(* IEC 61131-3 sources: TA/Tests/RetainTest/OLD/FBtest (part 4) *)

    ARRAY_LWORD_OUT_AUTO_2[0] := ARRAY_LWORD_OUT_AUTO_1[0];
    ARRAY_LWORD_OUT_AUTO_2[1] := ARRAY_LWORD_OUT_AUTO_1[1];
    ARRAY_LWORD_OUT_AUTO_2[2] := ARRAY_LWORD_OUT_AUTO_1[2];
    ARRAY_LWORD_OUT_AUTO_2[3] := ARRAY_LWORD_OUT_AUTO_1[3];
    ARRAY_LWORD_OUT_AUTO_2[4] := ARRAY_LWORD_OUT_AUTO_1[4];
    ARRAY_LWORD_OUT_AUTO_2[5] := ARRAY_LWORD_OUT_AUTO_1[5];
    ARRAY_LWORD_OUT_AUTO_2[6] := ARRAY_LWORD_OUT_AUTO_1[6];
    ARRAY_LWORD_OUT_AUTO_2[7] := ARRAY_LWORD_OUT_AUTO_1[7];
    ARRAY_LWORD_OUT_AUTO_2[8] := ARRAY_LWORD_OUT_AUTO_1[8];
    ARRAY_LWORD_OUT_AUTO_2[9] := ARRAY_LWORD_OUT_AUTO_1[9];

    ARRAY_REAL_OUT_AUTO_2[0] := ARRAY_REAL_OUT_AUTO_1[0];
    ARRAY_REAL_OUT_AUTO_2[1] := ARRAY_REAL_OUT_AUTO_1[1];
    ARRAY_REAL_OUT_AUTO_2[2] := ARRAY_REAL_OUT_AUTO_1[2];
    ARRAY_REAL_OUT_AUTO_2[3] := ARRAY_REAL_OUT_AUTO_1[3];
    ARRAY_REAL_OUT_AUTO_2[4] := ARRAY_REAL_OUT_AUTO_1[4];
    ARRAY_REAL_OUT_AUTO_2[5] := ARRAY_REAL_OUT_AUTO_1[5];
    ARRAY_REAL_OUT_AUTO_2[6] := ARRAY_REAL_OUT_AUTO_1[6];
    ARRAY_REAL_OUT_AUTO_2[7] := ARRAY_REAL_OUT_AUTO_1[7];
    ARRAY_REAL_OUT_AUTO_2[8] := ARRAY_REAL_OUT_AUTO_1[8];
    ARRAY_REAL_OUT_AUTO_2[9] := ARRAY_REAL_OUT_AUTO_1[9];

    ARRAY_SINT_OUT_AUTO_2[0] := ARRAY_SINT_OUT_AUTO_1[0];
    ARRAY_SINT_OUT_AUTO_2[1] := ARRAY_SINT_OUT_AUTO_1[1];
    ARRAY_SINT_OUT_AUTO_2[2] := ARRAY_SINT_OUT_AUTO_1[2];
    ARRAY_SINT_OUT_AUTO_2[3] := ARRAY_SINT_OUT_AUTO_1[3];
    ARRAY_SINT_OUT_AUTO_2[4] := ARRAY_SINT_OUT_AUTO_1[4];
    ARRAY_SINT_OUT_AUTO_2[5] := ARRAY_SINT_OUT_AUTO_1[5];
    ARRAY_SINT_OUT_AUTO_2[6] := ARRAY_SINT_OUT_AUTO_1[6];
    ARRAY_SINT_OUT_AUTO_2[7] := ARRAY_SINT_OUT_AUTO_1[7];
    ARRAY_SINT_OUT_AUTO_2[8] := ARRAY_SINT_OUT_AUTO_1[8];
    ARRAY_SINT_OUT_AUTO_2[9] := ARRAY_SINT_OUT_AUTO_1[9];

    ARRAY_STRING_OUT_AUTO_2[0] := ARRAY_STRING_OUT_AUTO_1[0];
    ARRAY_STRING_OUT_AUTO_2[1] := ARRAY_STRING_OUT_AUTO_1[1];
    ARRAY_STRING_OUT_AUTO_2[2] := ARRAY_STRING_OUT_AUTO_1[2];
    ARRAY_STRING_OUT_AUTO_2[3] := ARRAY_STRING_OUT_AUTO_1[3];
    ARRAY_STRING_OUT_AUTO_2[4] := ARRAY_STRING_OUT_AUTO_1[4];
    ARRAY_STRING_OUT_AUTO_2[5] := ARRAY_STRING_OUT_AUTO_1[5];
    ARRAY_STRING_OUT_AUTO_2[6] := ARRAY_STRING_OUT_AUTO_1[6];
    ARRAY_STRING_OUT_AUTO_2[7] := ARRAY_STRING_OUT_AUTO_1[7];
    ARRAY_STRING_OUT_AUTO_2[8] := ARRAY_STRING_OUT_AUTO_1[8];
    ARRAY_STRING_OUT_AUTO_2[9] := ARRAY_STRING_OUT_AUTO_1[9];

    ARRAY_TIME_OUT_AUTO_2[0] := ARRAY_TIME_OUT_AUTO_1[0];
    ARRAY_TIME_OUT_AUTO_2[1] := ARRAY_TIME_OUT_AUTO_1[1];
    ARRAY_TIME_OUT_AUTO_2[2] := ARRAY_TIME_OUT_AUTO_1[2];
    ARRAY_TIME_OUT_AUTO_2[3] := ARRAY_TIME_OUT_AUTO_1[3];
    ARRAY_TIME_OUT_AUTO_2[4] := ARRAY_TIME_OUT_AUTO_1[4];
    ARRAY_TIME_OUT_AUTO_2[5] := ARRAY_TIME_OUT_AUTO_1[5];
    ARRAY_TIME_OUT_AUTO_2[6] := ARRAY_TIME_OUT_AUTO_1[6];
    ARRAY_TIME_OUT_AUTO_2[7] := ARRAY_TIME_OUT_AUTO_1[7];
    ARRAY_TIME_OUT_AUTO_2[8] := ARRAY_TIME_OUT_AUTO_1[8];
    ARRAY_TIME_OUT_AUTO_2[9] := ARRAY_TIME_OUT_AUTO_1[9];

    ARRAY_UDINT_OUT_AUTO_2[0] := ARRAY_UDINT_OUT_AUTO_1[0];
    ARRAY_UDINT_OUT_AUTO_2[1] := ARRAY_UDINT_OUT_AUTO_1[1];
    ARRAY_UDINT_OUT_AUTO_2[2] := ARRAY_UDINT_OUT_AUTO_1[2];
    ARRAY_UDINT_OUT_AUTO_2[3] := ARRAY_UDINT_OUT_AUTO_1[3];
    ARRAY_UDINT_OUT_AUTO_2[4] := ARRAY_UDINT_OUT_AUTO_1[4];
    ARRAY_UDINT_OUT_AUTO_2[5] := ARRAY_UDINT_OUT_AUTO_1[5];
    ARRAY_UDINT_OUT_AUTO_2[6] := ARRAY_UDINT_OUT_AUTO_1[6];
    ARRAY_UDINT_OUT_AUTO_2[7] := ARRAY_UDINT_OUT_AUTO_1[7];
    ARRAY_UDINT_OUT_AUTO_2[8] := ARRAY_UDINT_OUT_AUTO_1[6];
    ARRAY_UDINT_OUT_AUTO_2[9] := ARRAY_UDINT_OUT_AUTO_1[7];

    ARRAY_UINT_OUT_AUTO_2[0] := ARRAY_UINT_OUT_AUTO_1[0];
    ARRAY_UINT_OUT_AUTO_2[1] := ARRAY_UINT_OUT_AUTO_1[1];
    ARRAY_UINT_OUT_AUTO_2[2] := ARRAY_UINT_OUT_AUTO_1[2];
    ARRAY_UINT_OUT_AUTO_2[3] := ARRAY_UINT_OUT_AUTO_1[3];
    ARRAY_UINT_OUT_AUTO_2[4] := ARRAY_UINT_OUT_AUTO_1[4];
    ARRAY_UINT_OUT_AUTO_2[5] := ARRAY_UINT_OUT_AUTO_1[5];
    ARRAY_UINT_OUT_AUTO_2[6] := ARRAY_UINT_OUT_AUTO_1[6];
    ARRAY_UINT_OUT_AUTO_2[7] := ARRAY_UINT_OUT_AUTO_1[7];
    ARRAY_UINT_OUT_AUTO_2[8] := ARRAY_UINT_OUT_AUTO_1[8];
    ARRAY_UINT_OUT_AUTO_2[9] := ARRAY_UINT_OUT_AUTO_1[9];

    ARRAY_ULINT_OUT_AUTO_2[0] := ARRAY_ULINT_OUT_AUTO_1[0];
    ARRAY_ULINT_OUT_AUTO_2[1] := ARRAY_ULINT_OUT_AUTO_1[1];
    ARRAY_ULINT_OUT_AUTO_2[2] := ARRAY_ULINT_OUT_AUTO_1[2];
    ARRAY_ULINT_OUT_AUTO_2[3] := ARRAY_ULINT_OUT_AUTO_1[3];
    ARRAY_ULINT_OUT_AUTO_2[4] := ARRAY_ULINT_OUT_AUTO_1[4];
    ARRAY_ULINT_OUT_AUTO_2[5] := ARRAY_ULINT_OUT_AUTO_1[5];
    ARRAY_ULINT_OUT_AUTO_2[6] := ARRAY_ULINT_OUT_AUTO_1[6];
    ARRAY_ULINT_OUT_AUTO_2[7] := ARRAY_ULINT_OUT_AUTO_1[7];
    ARRAY_ULINT_OUT_AUTO_2[8] := ARRAY_ULINT_OUT_AUTO_1[8];
    ARRAY_ULINT_OUT_AUTO_2[9] := ARRAY_ULINT_OUT_AUTO_1[9];

    ARRAY_USINT_OUT_AUTO_2[0] := ARRAY_USINT_OUT_AUTO_1[0];
    ARRAY_USINT_OUT_AUTO_2[1] := ARRAY_USINT_OUT_AUTO_1[1];
    ARRAY_USINT_OUT_AUTO_2[2] := ARRAY_USINT_OUT_AUTO_1[2];
    ARRAY_USINT_OUT_AUTO_2[3] := ARRAY_USINT_OUT_AUTO_1[3];
    ARRAY_USINT_OUT_AUTO_2[4] := ARRAY_USINT_OUT_AUTO_1[4];
    ARRAY_USINT_OUT_AUTO_2[5] := ARRAY_USINT_OUT_AUTO_1[5];
    ARRAY_USINT_OUT_AUTO_2[6] := ARRAY_USINT_OUT_AUTO_1[6];
    ARRAY_USINT_OUT_AUTO_2[7] := ARRAY_USINT_OUT_AUTO_1[7];
    ARRAY_USINT_OUT_AUTO_2[8] := ARRAY_USINT_OUT_AUTO_1[8];
    ARRAY_USINT_OUT_AUTO_2[9] := ARRAY_USINT_OUT_AUTO_1[9];

    ARRAY_WORD_OUT_AUTO_2[0] := ARRAY_WORD_OUT_AUTO_1[0];
    ARRAY_WORD_OUT_AUTO_2[1] := ARRAY_WORD_OUT_AUTO_1[1];
    ARRAY_WORD_OUT_AUTO_2[2] := ARRAY_WORD_OUT_AUTO_1[2];
    ARRAY_WORD_OUT_AUTO_2[3] := ARRAY_WORD_OUT_AUTO_1[3];
    ARRAY_WORD_OUT_AUTO_2[4] := ARRAY_WORD_OUT_AUTO_1[4];
    ARRAY_WORD_OUT_AUTO_2[5] := ARRAY_WORD_OUT_AUTO_1[5];
    ARRAY_WORD_OUT_AUTO_2[6] := ARRAY_WORD_OUT_AUTO_1[6];
    ARRAY_WORD_OUT_AUTO_2[7] := ARRAY_WORD_OUT_AUTO_1[7];
    ARRAY_WORD_OUT_AUTO_2[8] := ARRAY_WORD_OUT_AUTO_1[8];
    ARRAY_WORD_OUT_AUTO_2[9] := ARRAY_WORD_OUT_AUTO_1[9];

END_IF;

END_FUNCTION_BLOCK

(* ---- FB_FB_SIMPLE_TYPE.st ---- *)
FUNCTION_BLOCK FB_FB_SIMPLE_TYPE

// ЗАПУСК ФБ
FB_SIMPLE_TYPE_RETAIN.TRIGGER_IMP := TRIGGER_IMP;
FB_SIMPLE_TYPE_NON_RETAIN.TRIGGER_IMP := TRIGGER_IMP;
FB_SIMPLE_TYPE_AUTO.TRIGGER_IMP := TRIGGER_IMP;

FB_SIMPLE_TYPE_RETAIN(.BOOL_IN, .BYTE_IN, .DATE_IN, .DINT_IN, .DWORD_IN, .INT_IN, .LINT_IN, .LREAL_IN, .LWORD_IN, .REAL_IN, .SINT_IN, .STRING_IN, .TIME_IN, .UDINT_IN, .UINT_IN, .ULINT_IN, .USINT_IN, .WORD_IN, .TRIGGER_IMP);
FB_SIMPLE_TYPE_NON_RETAIN(.BOOL_IN, .BYTE_IN, .DATE_IN, .DINT_IN, .DWORD_IN, .INT_IN, .LINT_IN, .LREAL_IN, .LWORD_IN, .REAL_IN, .SINT_IN, .STRING_IN, .TIME_IN, .UDINT_IN, .UINT_IN, .ULINT_IN, .USINT_IN, .WORD_IN, .TRIGGER_IMP);
FB_SIMPLE_TYPE_AUTO(.BOOL_IN, .BYTE_IN, .DATE_IN, .DINT_IN, .DWORD_IN, .INT_IN, .LINT_IN, .LREAL_IN, .LWORD_IN, .REAL_IN, .SINT_IN, .STRING_IN, .TIME_IN, .UDINT_IN, .UINT_IN, .ULINT_IN, .USINT_IN, .WORD_IN, .TRIGGER_IMP);

IF TRIGGER_IMP THEN

    FB_SIMPLE_TYPE_RETAIN.BOOL_IN := NOT FB_SIMPLE_TYPE_RETAIN.BOOL_IN;
    FB_SIMPLE_TYPE_RETAIN.BYTE_IN := FB_SIMPLE_TYPE_RETAIN.BYTE_IN + 1;
    FB_SIMPLE_TYPE_RETAIN.DATE_IN := ANY_TO_DATE(1445385600 + FB_SIMPLE_TYPE_RETAIN.DINT_IN * 86400);
    FB_SIMPLE_TYPE_RETAIN.DINT_IN := FB_SIMPLE_TYPE_RETAIN.DINT_IN + 1;
    FB_SIMPLE_TYPE_RETAIN.DWORD_IN := FB_SIMPLE_TYPE_RETAIN.DWORD_IN + 1;
    FB_SIMPLE_TYPE_RETAIN.INT_IN := FB_SIMPLE_TYPE_RETAIN.INT_IN + 1;
    FB_SIMPLE_TYPE_RETAIN.LINT_IN := FB_SIMPLE_TYPE_RETAIN.LINT_IN + 1;
    FB_SIMPLE_TYPE_RETAIN.LREAL_IN := FB_SIMPLE_TYPE_RETAIN.LREAL_IN + 1.1;
    FB_SIMPLE_TYPE_RETAIN.LWORD_IN := FB_SIMPLE_TYPE_RETAIN.LWORD_IN + 1;
    FB_SIMPLE_TYPE_RETAIN.REAL_IN := FB_SIMPLE_TYPE_RETAIN.REAL_IN + 1.1;
    FB_SIMPLE_TYPE_RETAIN.SINT_IN := FB_SIMPLE_TYPE_RETAIN.SINT_IN + 1;
    FB_SIMPLE_TYPE_RETAIN.STRING_IN := ANY_TO_STRING(FB_SIMPLE_TYPE_RETAIN.DINT_IN) + ' ' + ANY_TO_STRING(FB_SIMPLE_TYPE_RETAIN.TIME_IN);
    FB_SIMPLE_TYPE_RETAIN.TIME_IN := FB_SIMPLE_TYPE_RETAIN.TIME_IN + PULSE_TIME;
    FB_SIMPLE_TYPE_RETAIN.UDINT_IN := FB_SIMPLE_TYPE_RETAIN.UDINT_IN + 1;
    FB_SIMPLE_TYPE_RETAIN.UINT_IN := FB_SIMPLE_TYPE_RETAIN.UINT_IN + 1;
    FB_SIMPLE_TYPE_RETAIN.ULINT_IN := FB_SIMPLE_TYPE_RETAIN.ULINT_IN + 1;
    FB_SIMPLE_TYPE_RETAIN.USINT_IN := FB_SIMPLE_TYPE_RETAIN.USINT_IN + 1;
    FB_SIMPLE_TYPE_RETAIN.WORD_IN := FB_SIMPLE_TYPE_RETAIN.WORD_IN + 1;

    FB_SIMPLE_TYPE_RETAIN.BOOL_IN := NOT FB_SIMPLE_TYPE_RETAIN.BOOL_IN;
    FB_SIMPLE_TYPE_RETAIN.BYTE_IN := FB_SIMPLE_TYPE_RETAIN.BYTE_IN + 1;
    FB_SIMPLE_TYPE_RETAIN.DATE_IN := ANY_TO_DATE(1445385600 + FB_SIMPLE_TYPE_RETAIN.DINT_IN * 86400);
    FB_SIMPLE_TYPE_RETAIN.DINT_IN := FB_SIMPLE_TYPE_RETAIN.DINT_IN + 1;
    FB_SIMPLE_TYPE_RETAIN.DWORD_IN := FB_SIMPLE_TYPE_RETAIN.DWORD_IN + 1;
    FB_SIMPLE_TYPE_RETAIN.INT_IN := FB_SIMPLE_TYPE_RETAIN.INT_IN + 1;
    FB_SIMPLE_TYPE_RETAIN.LINT_IN := FB_SIMPLE_TYPE_RETAIN.LINT_IN + 1;
    FB_SIMPLE_TYPE_RETAIN.LREAL_IN := FB_SIMPLE_TYPE_RETAIN.LREAL_IN + 1.1;
    FB_SIMPLE_TYPE_RETAIN.LWORD_IN := FB_SIMPLE_TYPE_RETAIN.LWORD_IN + 1;
    FB_SIMPLE_TYPE_RETAIN.REAL_IN := FB_SIMPLE_TYPE_RETAIN.REAL_IN + 1.1;
    FB_SIMPLE_TYPE_RETAIN.SINT_IN := FB_SIMPLE_TYPE_RETAIN.SINT_IN + 1;
    FB_SIMPLE_TYPE_RETAIN.STRING_IN := ANY_TO_STRING(FB_SIMPLE_TYPE_RETAIN.DINT_IN) + ' ' + ANY_TO_STRING(FB_SIMPLE_TYPE_RETAIN.TIME_IN);
    FB_SIMPLE_TYPE_RETAIN.TIME_IN := FB_SIMPLE_TYPE_RETAIN.TIME_IN + PULSE_TIME;
    FB_SIMPLE_TYPE_RETAIN.UDINT_IN := FB_SIMPLE_TYPE_RETAIN.UDINT_IN + 1;
    FB_SIMPLE_TYPE_RETAIN.UINT_IN := FB_SIMPLE_TYPE_RETAIN.UINT_IN + 1;
    FB_SIMPLE_TYPE_RETAIN.ULINT_IN := FB_SIMPLE_TYPE_RETAIN.ULINT_IN + 1;
    FB_SIMPLE_TYPE_RETAIN.USINT_IN := FB_SIMPLE_TYPE_RETAIN.USINT_IN + 1;
    FB_SIMPLE_TYPE_RETAIN.WORD_IN := FB_SIMPLE_TYPE_RETAIN.WORD_IN + 1;

    FB_SIMPLE_TYPE_RETAIN.BOOL_IN := NOT FB_SIMPLE_TYPE_RETAIN.BOOL_IN;
    FB_SIMPLE_TYPE_RETAIN.BYTE_IN := FB_SIMPLE_TYPE_RETAIN.BYTE_IN + 1;
    FB_SIMPLE_TYPE_RETAIN.DATE_IN := ANY_TO_DATE(1445385600 + FB_SIMPLE_TYPE_RETAIN.DINT_IN * 86400);
    FB_SIMPLE_TYPE_RETAIN.DINT_IN := FB_SIMPLE_TYPE_RETAIN.DINT_IN + 1;
    FB_SIMPLE_TYPE_RETAIN.DWORD_IN := FB_SIMPLE_TYPE_RETAIN.DWORD_IN + 1;
    FB_SIMPLE_TYPE_RETAIN.INT_IN := FB_SIMPLE_TYPE_RETAIN.INT_IN + 1;
    FB_SIMPLE_TYPE_RETAIN.LINT_IN := FB_SIMPLE_TYPE_RETAIN.LINT_IN + 1;
    FB_SIMPLE_TYPE_RETAIN.LREAL_IN := FB_SIMPLE_TYPE_RETAIN.LREAL_IN + 1.1;
    FB_SIMPLE_TYPE_RETAIN.LWORD_IN := FB_SIMPLE_TYPE_RETAIN.LWORD_IN + 1;
    FB_SIMPLE_TYPE_RETAIN.REAL_IN := FB_SIMPLE_TYPE_RETAIN.REAL_IN + 1.1;
    FB_SIMPLE_TYPE_RETAIN.SINT_IN := FB_SIMPLE_TYPE_RETAIN.SINT_IN + 1;
    FB_SIMPLE_TYPE_RETAIN.STRING_IN := ANY_TO_STRING(FB_SIMPLE_TYPE_RETAIN.DINT_IN) + ' ' + ANY_TO_STRING(FB_SIMPLE_TYPE_RETAIN.TIME_IN);
    FB_SIMPLE_TYPE_RETAIN.TIME_IN := FB_SIMPLE_TYPE_RETAIN.TIME_IN + PULSE_TIME;
    FB_SIMPLE_TYPE_RETAIN.UDINT_IN := FB_SIMPLE_TYPE_RETAIN.UDINT_IN + 1;
    FB_SIMPLE_TYPE_RETAIN.UINT_IN := FB_SIMPLE_TYPE_RETAIN.UINT_IN + 1;
    FB_SIMPLE_TYPE_RETAIN.ULINT_IN := FB_SIMPLE_TYPE_RETAIN.ULINT_IN + 1;
    FB_SIMPLE_TYPE_RETAIN.USINT_IN := FB_SIMPLE_TYPE_RETAIN.USINT_IN + 1;
    FB_SIMPLE_TYPE_RETAIN.WORD_IN := FB_SIMPLE_TYPE_RETAIN.WORD_IN + 1;

    FB_SIMPLE_TYPE_NON_RETAIN.BOOL_IN := NOT FB_SIMPLE_TYPE_NON_RETAIN.BOOL_IN;
    FB_SIMPLE_TYPE_NON_RETAIN.BYTE_IN := FB_SIMPLE_TYPE_NON_RETAIN.BYTE_IN + 1;
    FB_SIMPLE_TYPE_NON_RETAIN.DATE_IN := ANY_TO_DATE(1445385600 + FB_SIMPLE_TYPE_NON_RETAIN.DINT_IN * 86400);
    FB_SIMPLE_TYPE_NON_RETAIN.DINT_IN := FB_SIMPLE_TYPE_NON_RETAIN.DINT_IN + 1;
    FB_SIMPLE_TYPE_NON_RETAIN.DWORD_IN := FB_SIMPLE_TYPE_NON_RETAIN.DWORD_IN + 1;
    FB_SIMPLE_TYPE_NON_RETAIN.INT_IN := FB_SIMPLE_TYPE_NON_RETAIN.INT_IN + 1;
    FB_SIMPLE_TYPE_NON_RETAIN.LINT_IN := FB_SIMPLE_TYPE_NON_RETAIN.LINT_IN + 1;
    FB_SIMPLE_TYPE_NON_RETAIN.LREAL_IN := FB_SIMPLE_TYPE_NON_RETAIN.LREAL_IN + 1.1;
    FB_SIMPLE_TYPE_NON_RETAIN.LWORD_IN := FB_SIMPLE_TYPE_NON_RETAIN.LWORD_IN + 1;
    FB_SIMPLE_TYPE_NON_RETAIN.REAL_IN := FB_SIMPLE_TYPE_NON_RETAIN.REAL_IN + 1.1;
    FB_SIMPLE_TYPE_NON_RETAIN.SINT_IN := FB_SIMPLE_TYPE_NON_RETAIN.SINT_IN + 1;
    FB_SIMPLE_TYPE_NON_RETAIN.STRING_IN := ANY_TO_STRING(FB_SIMPLE_TYPE_NON_RETAIN.DINT_IN) + ' ' + ANY_TO_STRING(FB_SIMPLE_TYPE_NON_RETAIN.TIME_IN);
    FB_SIMPLE_TYPE_NON_RETAIN.TIME_IN := FB_SIMPLE_TYPE_NON_RETAIN.TIME_IN + PULSE_TIME;
    FB_SIMPLE_TYPE_NON_RETAIN.UDINT_IN := FB_SIMPLE_TYPE_NON_RETAIN.UDINT_IN + 1;
    FB_SIMPLE_TYPE_NON_RETAIN.UINT_IN := FB_SIMPLE_TYPE_NON_RETAIN.UINT_IN + 1;
    FB_SIMPLE_TYPE_NON_RETAIN.ULINT_IN := FB_SIMPLE_TYPE_NON_RETAIN.ULINT_IN + 1;
    FB_SIMPLE_TYPE_NON_RETAIN.USINT_IN := FB_SIMPLE_TYPE_NON_RETAIN.USINT_IN + 1;
    FB_SIMPLE_TYPE_NON_RETAIN.WORD_IN := FB_SIMPLE_TYPE_NON_RETAIN.WORD_IN + 1;

    FB_SIMPLE_TYPE_NON_RETAIN.BOOL_IN := NOT FB_SIMPLE_TYPE_NON_RETAIN.BOOL_IN;
    FB_SIMPLE_TYPE_NON_RETAIN.BYTE_IN := FB_SIMPLE_TYPE_NON_RETAIN.BYTE_IN + 1;
    FB_SIMPLE_TYPE_NON_RETAIN.DATE_IN := ANY_TO_DATE(1445385600 + FB_SIMPLE_TYPE_NON_RETAIN.DINT_IN * 86400);
    FB_SIMPLE_TYPE_NON_RETAIN.DINT_IN := FB_SIMPLE_TYPE_NON_RETAIN.DINT_IN + 1;
    FB_SIMPLE_TYPE_NON_RETAIN.DWORD_IN := FB_SIMPLE_TYPE_NON_RETAIN.DWORD_IN + 1;
    FB_SIMPLE_TYPE_NON_RETAIN.INT_IN := FB_SIMPLE_TYPE_NON_RETAIN.INT_IN + 1;
    FB_SIMPLE_TYPE_NON_RETAIN.LINT_IN := FB_SIMPLE_TYPE_NON_RETAIN.LINT_IN + 1;
    FB_SIMPLE_TYPE_NON_RETAIN.LREAL_IN := FB_SIMPLE_TYPE_NON_RETAIN.LREAL_IN + 1.1;
    FB_SIMPLE_TYPE_NON_RETAIN.LWORD_IN := FB_SIMPLE_TYPE_NON_RETAIN.LWORD_IN + 1;
    FB_SIMPLE_TYPE_NON_RETAIN.REAL_IN := FB_SIMPLE_TYPE_NON_RETAIN.REAL_IN + 1.1;
    FB_SIMPLE_TYPE_NON_RETAIN.SINT_IN := FB_SIMPLE_TYPE_NON_RETAIN.SINT_IN + 1;
    FB_SIMPLE_TYPE_NON_RETAIN.STRING_IN := ANY_TO_STRING(FB_SIMPLE_TYPE_NON_RETAIN.DINT_IN) + ' ' + ANY_TO_STRING(FB_SIMPLE_TYPE_NON_RETAIN.TIME_IN);
    FB_SIMPLE_TYPE_NON_RETAIN.TIME_IN := FB_SIMPLE_TYPE_NON_RETAIN.TIME_IN + PULSE_TIME;
    FB_SIMPLE_TYPE_NON_RETAIN.UDINT_IN := FB_SIMPLE_TYPE_NON_RETAIN.UDINT_IN + 1;
    FB_SIMPLE_TYPE_NON_RETAIN.UINT_IN := FB_SIMPLE_TYPE_NON_RETAIN.UINT_IN + 1;
    FB_SIMPLE_TYPE_NON_RETAIN.ULINT_IN := FB_SIMPLE_TYPE_NON_RETAIN.ULINT_IN + 1;
    FB_SIMPLE_TYPE_NON_RETAIN.USINT_IN := FB_SIMPLE_TYPE_NON_RETAIN.USINT_IN + 1;
    FB_SIMPLE_TYPE_NON_RETAIN.WORD_IN := FB_SIMPLE_TYPE_NON_RETAIN.WORD_IN + 1;

    FB_SIMPLE_TYPE_NON_RETAIN.BOOL_IN := NOT FB_SIMPLE_TYPE_NON_RETAIN.BOOL_IN;
    FB_SIMPLE_TYPE_NON_RETAIN.BYTE_IN := FB_SIMPLE_TYPE_NON_RETAIN.BYTE_IN + 1;
    FB_SIMPLE_TYPE_NON_RETAIN.DATE_IN := ANY_TO_DATE(1445385600 + FB_SIMPLE_TYPE_NON_RETAIN.DINT_IN * 86400);
    FB_SIMPLE_TYPE_NON_RETAIN.DINT_IN := FB_SIMPLE_TYPE_NON_RETAIN.DINT_IN + 1;
    FB_SIMPLE_TYPE_NON_RETAIN.DWORD_IN := FB_SIMPLE_TYPE_NON_RETAIN.DWORD_IN + 1;
    FB_SIMPLE_TYPE_NON_RETAIN.INT_IN := FB_SIMPLE_TYPE_NON_RETAIN.INT_IN + 1;
    FB_SIMPLE_TYPE_NON_RETAIN.LINT_IN := FB_SIMPLE_TYPE_NON_RETAIN.LINT_IN + 1;
    FB_SIMPLE_TYPE_NON_RETAIN.LREAL_IN := FB_SIMPLE_TYPE_NON_RETAIN.LREAL_IN + 1.1;
    FB_SIMPLE_TYPE_NON_RETAIN.LWORD_IN := FB_SIMPLE_TYPE_NON_RETAIN.LWORD_IN + 1;
    FB_SIMPLE_TYPE_NON_RETAIN.REAL_IN := FB_SIMPLE_TYPE_NON_RETAIN.REAL_IN + 1.1;
    FB_SIMPLE_TYPE_NON_RETAIN.SINT_IN := FB_SIMPLE_TYPE_NON_RETAIN.SINT_IN + 1;
    FB_SIMPLE_TYPE_NON_RETAIN.STRING_IN := ANY_TO_STRING(FB_SIMPLE_TYPE_NON_RETAIN.DINT_IN) + ' ' + ANY_TO_STRING(FB_SIMPLE_TYPE_NON_RETAIN.TIME_IN);
    FB_SIMPLE_TYPE_NON_RETAIN.TIME_IN := FB_SIMPLE_TYPE_NON_RETAIN.TIME_IN + PULSE_TIME;
    FB_SIMPLE_TYPE_NON_RETAIN.UDINT_IN := FB_SIMPLE_TYPE_NON_RETAIN.UDINT_IN + 1;
    FB_SIMPLE_TYPE_NON_RETAIN.UINT_IN := FB_SIMPLE_TYPE_NON_RETAIN.UINT_IN + 1;
    FB_SIMPLE_TYPE_NON_RETAIN.ULINT_IN := FB_SIMPLE_TYPE_NON_RETAIN.ULINT_IN + 1;
    FB_SIMPLE_TYPE_NON_RETAIN.USINT_IN := FB_SIMPLE_TYPE_NON_RETAIN.USINT_IN + 1;
    FB_SIMPLE_TYPE_NON_RETAIN.WORD_IN := FB_SIMPLE_TYPE_NON_RETAIN.WORD_IN + 1;

    FB_SIMPLE_TYPE_AUTO.BOOL_IN := NOT FB_SIMPLE_TYPE_AUTO.BOOL_IN;
    FB_SIMPLE_TYPE_AUTO.BYTE_IN := FB_SIMPLE_TYPE_AUTO.BYTE_IN + 1;
    FB_SIMPLE_TYPE_AUTO.DATE_IN := ANY_TO_DATE(1445385600 + FB_SIMPLE_TYPE_AUTO.DINT_IN * 86400);
    FB_SIMPLE_TYPE_AUTO.DINT_IN := FB_SIMPLE_TYPE_AUTO.DINT_IN + 1;
    FB_SIMPLE_TYPE_AUTO.DWORD_IN := FB_SIMPLE_TYPE_AUTO.DWORD_IN + 1;
    FB_SIMPLE_TYPE_AUTO.INT_IN := FB_SIMPLE_TYPE_AUTO.INT_IN + 1;
    FB_SIMPLE_TYPE_AUTO.LINT_IN := FB_SIMPLE_TYPE_AUTO.LINT_IN + 1;
    FB_SIMPLE_TYPE_AUTO.LREAL_IN := FB_SIMPLE_TYPE_AUTO.LREAL_IN + 1.1;
    FB_SIMPLE_TYPE_AUTO.LWORD_IN := FB_SIMPLE_TYPE_AUTO.LWORD_IN + 1;
    FB_SIMPLE_TYPE_AUTO.REAL_IN := FB_SIMPLE_TYPE_AUTO.REAL_IN + 1.1;
    FB_SIMPLE_TYPE_AUTO.SINT_IN := FB_SIMPLE_TYPE_AUTO.SINT_IN + 1;
    FB_SIMPLE_TYPE_AUTO.STRING_IN := ANY_TO_STRING(FB_SIMPLE_TYPE_AUTO.DINT_IN) + ' ' + ANY_TO_STRING(FB_SIMPLE_TYPE_AUTO.TIME_IN);
    FB_SIMPLE_TYPE_AUTO.TIME_IN := FB_SIMPLE_TYPE_AUTO.TIME_IN + PULSE_TIME;
    FB_SIMPLE_TYPE_AUTO.UDINT_IN := FB_SIMPLE_TYPE_AUTO.UDINT_IN + 1;
    FB_SIMPLE_TYPE_AUTO.UINT_IN := FB_SIMPLE_TYPE_AUTO.UINT_IN + 1;
    FB_SIMPLE_TYPE_AUTO.ULINT_IN := FB_SIMPLE_TYPE_AUTO.ULINT_IN + 1;
    FB_SIMPLE_TYPE_AUTO.USINT_IN := FB_SIMPLE_TYPE_AUTO.USINT_IN + 1;
    FB_SIMPLE_TYPE_AUTO.WORD_IN := FB_SIMPLE_TYPE_AUTO.WORD_IN + 1;

    FB_SIMPLE_TYPE_AUTO.BOOL_IN := NOT FB_SIMPLE_TYPE_AUTO.BOOL_IN;
    FB_SIMPLE_TYPE_AUTO.BYTE_IN := FB_SIMPLE_TYPE_AUTO.BYTE_IN + 1;
    FB_SIMPLE_TYPE_AUTO.DATE_IN := ANY_TO_DATE(1445385600 + FB_SIMPLE_TYPE_AUTO.DINT_IN * 86400);
    FB_SIMPLE_TYPE_AUTO.DINT_IN := FB_SIMPLE_TYPE_AUTO.DINT_IN + 1;
    FB_SIMPLE_TYPE_AUTO.DWORD_IN := FB_SIMPLE_TYPE_AUTO.DWORD_IN + 1;
    FB_SIMPLE_TYPE_AUTO.INT_IN := FB_SIMPLE_TYPE_AUTO.INT_IN + 1;
    FB_SIMPLE_TYPE_AUTO.LINT_IN := FB_SIMPLE_TYPE_AUTO.LINT_IN + 1;
    FB_SIMPLE_TYPE_AUTO.LREAL_IN := FB_SIMPLE_TYPE_AUTO.LREAL_IN + 1.1;
    FB_SIMPLE_TYPE_AUTO.LWORD_IN := FB_SIMPLE_TYPE_AUTO.LWORD_IN + 1;
    FB_SIMPLE_TYPE_AUTO.REAL_IN := FB_SIMPLE_TYPE_AUTO.REAL_IN + 1.1;
    FB_SIMPLE_TYPE_AUTO.SINT_IN := FB_SIMPLE_TYPE_AUTO.SINT_IN + 1;
    FB_SIMPLE_TYPE_AUTO.STRING_IN := ANY_TO_STRING(FB_SIMPLE_TYPE_AUTO.DINT_IN) + ' ' + ANY_TO_STRING(FB_SIMPLE_TYPE_AUTO.TIME_IN);
    FB_SIMPLE_TYPE_AUTO.TIME_IN := FB_SIMPLE_TYPE_AUTO.TIME_IN + PULSE_TIME;
    FB_SIMPLE_TYPE_AUTO.UDINT_IN := FB_SIMPLE_TYPE_AUTO.UDINT_IN + 1;
    FB_SIMPLE_TYPE_AUTO.UINT_IN := FB_SIMPLE_TYPE_AUTO.UINT_IN + 1;
    FB_SIMPLE_TYPE_AUTO.ULINT_IN := FB_SIMPLE_TYPE_AUTO.ULINT_IN + 1;
    FB_SIMPLE_TYPE_AUTO.USINT_IN := FB_SIMPLE_TYPE_AUTO.USINT_IN + 1;
    FB_SIMPLE_TYPE_AUTO.WORD_IN := FB_SIMPLE_TYPE_AUTO.WORD_IN + 1;

    FB_SIMPLE_TYPE_AUTO.BOOL_IN := NOT FB_SIMPLE_TYPE_AUTO.BOOL_IN;
    FB_SIMPLE_TYPE_AUTO.BYTE_IN := FB_SIMPLE_TYPE_AUTO.BYTE_IN + 1;
    FB_SIMPLE_TYPE_AUTO.DATE_IN := ANY_TO_DATE(1445385600 + FB_SIMPLE_TYPE_AUTO.DINT_IN * 86400);
    FB_SIMPLE_TYPE_AUTO.DINT_IN := FB_SIMPLE_TYPE_AUTO.DINT_IN + 1;
    FB_SIMPLE_TYPE_AUTO.DWORD_IN := FB_SIMPLE_TYPE_AUTO.DWORD_IN + 1;
    FB_SIMPLE_TYPE_AUTO.INT_IN := FB_SIMPLE_TYPE_AUTO.INT_IN + 1;
    FB_SIMPLE_TYPE_AUTO.LINT_IN := FB_SIMPLE_TYPE_AUTO.LINT_IN + 1;
    FB_SIMPLE_TYPE_AUTO.LREAL_IN := FB_SIMPLE_TYPE_AUTO.LREAL_IN + 1.1;
    FB_SIMPLE_TYPE_AUTO.LWORD_IN := FB_SIMPLE_TYPE_AUTO.LWORD_IN + 1;
    FB_SIMPLE_TYPE_AUTO.REAL_IN := FB_SIMPLE_TYPE_AUTO.REAL_IN + 1.1;
    FB_SIMPLE_TYPE_AUTO.SINT_IN := FB_SIMPLE_TYPE_AUTO.SINT_IN + 1;
    FB_SIMPLE_TYPE_AUTO.STRING_IN := ANY_TO_STRING(FB_SIMPLE_TYPE_AUTO.DINT_IN) + ' ' + ANY_TO_STRING(FB_SIMPLE_TYPE_AUTO.TIME_IN);
    FB_SIMPLE_TYPE_AUTO.TIME_IN := FB_SIMPLE_TYPE_AUTO.TIME_IN + PULSE_TIME;
    FB_SIMPLE_TYPE_AUTO.UDINT_IN := FB_SIMPLE_TYPE_AUTO.UDINT_IN + 1;
    FB_SIMPLE_TYPE_AUTO.UINT_IN := FB_SIMPLE_TYPE_AUTO.UINT_IN + 1;
    FB_SIMPLE_TYPE_AUTO.ULINT_IN := FB_SIMPLE_TYPE_AUTO.ULINT_IN + 1;
    FB_SIMPLE_TYPE_AUTO.USINT_IN := FB_SIMPLE_TYPE_AUTO.USINT_IN + 1;
    FB_SIMPLE_TYPE_AUTO.WORD_IN := FB_SIMPLE_TYPE_AUTO.WORD_IN + 1;

END_IF;

END_FUNCTION_BLOCK

(* ---- FB_SIMPLE_TYPE_ALL.st ---- *)
FUNCTION_BLOCK FB_SIMPLE_TYPE_ALL

IF TRIGGER_IMP THEN

    // ЛОКАЛЬНЫЕ ПЕРЕМЕННЫЕ
    BOOL_LOCAL_RETAIN := NOT BOOL_LOCAL_RETAIN;
    BYTE_LOCAL_RETAIN := BYTE_LOCAL_RETAIN + 1;
    DATE_LOCAL_RETAIN := ANY_TO_DATE(1445385600 + DINT_LOCAL_RETAIN * 86400);
    DINT_LOCAL_RETAIN := DINT_LOCAL_RETAIN + 1;
    DWORD_LOCAL_RETAIN := DWORD_LOCAL_RETAIN + 1;
    INT_LOCAL_RETAIN := INT_LOCAL_RETAIN + 1;
    LINT_LOCAL_RETAIN := LINT_LOCAL_RETAIN + 1;
    LREAL_LOCAL_RETAIN := LREAL_LOCAL_RETAIN + 1.1;
    LWORD_LOCAL_RETAIN := LWORD_LOCAL_RETAIN + 1;
    REAL_LOCAL_RETAIN := REAL_LOCAL_RETAIN + 1.1;
    SINT_LOCAL_RETAIN := SINT_LOCAL_RETAIN + 1;
    STRING_LOCAL_RETAIN := ANY_TO_STRING(DINT_LOCAL_RETAIN) + ' ' + ANY_TO_STRING(TIME_LOCAL_RETAIN);
    TIME_LOCAL_RETAIN := TIME_LOCAL_RETAIN + T#10s;
    UDINT_LOCAL_RETAIN := UDINT_LOCAL_RETAIN + 1;
    UINT_LOCAL_RETAIN := UINT_LOCAL_RETAIN + 1;
    ULINT_LOCAL_RETAIN := ULINT_LOCAL_RETAIN + 1;
    USINT_LOCAL_RETAIN := USINT_LOCAL_RETAIN + 1;
    WORD_LOCAL_RETAIN := WORD_LOCAL_RETAIN + 1;

    BOOL_LOCAL_NON_RETAIN := NOT BOOL_LOCAL_NON_RETAIN;
    BYTE_LOCAL_NON_RETAIN := BYTE_LOCAL_NON_RETAIN + 1;
    DATE_LOCAL_NON_RETAIN := ANY_TO_DATE(1445385600 + DINT_LOCAL_NON_RETAIN * 86400);
    DINT_LOCAL_NON_RETAIN := DINT_LOCAL_NON_RETAIN + 1;
    DWORD_LOCAL_NON_RETAIN := DWORD_LOCAL_NON_RETAIN + 1;
    INT_LOCAL_NON_RETAIN := INT_LOCAL_NON_RETAIN + 1;
    LINT_LOCAL_NON_RETAIN := LINT_LOCAL_NON_RETAIN + 1;
    LREAL_LOCAL_NON_RETAIN := LREAL_LOCAL_NON_RETAIN + 1.1;
    LWORD_LOCAL_NON_RETAIN := LWORD_LOCAL_NON_RETAIN + 1;
    REAL_LOCAL_NON_RETAIN := REAL_LOCAL_NON_RETAIN + 1.1;
    SINT_LOCAL_NON_RETAIN := SINT_LOCAL_NON_RETAIN + 1;
    STRING_LOCAL_NON_RETAIN := ANY_TO_STRING(DINT_LOCAL_NON_RETAIN) + ' ' + ANY_TO_STRING(TIME_LOCAL_NON_RETAIN);
    TIME_LOCAL_NON_RETAIN := TIME_LOCAL_NON_RETAIN + T#10s;
    UDINT_LOCAL_NON_RETAIN := UDINT_LOCAL_NON_RETAIN + 1;
    UINT_LOCAL_NON_RETAIN := UINT_LOCAL_NON_RETAIN + 1;
    ULINT_LOCAL_NON_RETAIN := ULINT_LOCAL_NON_RETAIN + 1;
    USINT_LOCAL_NON_RETAIN := USINT_LOCAL_NON_RETAIN + 1;
    WORD_LOCAL_NON_RETAIN := WORD_LOCAL_NON_RETAIN + 1;

    BOOL_LOCAL_AUTO_1 := NOT BOOL_LOCAL_AUTO_1;
    BYTE_LOCAL_AUTO_1 := BYTE_LOCAL_AUTO_1 + 1;
    DATE_LOCAL_AUTO_1 := ANY_TO_DATE(1445385600 + DINT_LOCAL_AUTO_1 * 86400);
    DINT_LOCAL_AUTO_1 := DINT_LOCAL_AUTO_1 + 1;
    DWORD_LOCAL_AUTO_1 := DWORD_LOCAL_AUTO_1 + 1;
    INT_LOCAL_AUTO_1 := INT_LOCAL_AUTO_1 + 1;
    LINT_LOCAL_AUTO_1 := LINT_LOCAL_AUTO_1 + 1;
    LREAL_LOCAL_AUTO_1 := LREAL_LOCAL_AUTO_1 + 1.1;
    LWORD_LOCAL_AUTO_1 := LWORD_LOCAL_AUTO_1 + 1;
    REAL_LOCAL_AUTO_1 := REAL_LOCAL_AUTO_1 + 1.1;
    SINT_LOCAL_AUTO_1 := SINT_LOCAL_AUTO_1 + 1;
    STRING_LOCAL_AUTO_1 := ANY_TO_STRING(DINT_LOCAL_AUTO_1) + ' ' + ANY_TO_STRING(TIME_LOCAL_AUTO_1);
    TIME_LOCAL_AUTO_1 := TIME_LOCAL_AUTO_1 + T#10s;
    UDINT_LOCAL_AUTO_1 := UDINT_LOCAL_AUTO_1 + 1;
    UINT_LOCAL_AUTO_1 := UINT_LOCAL_AUTO_1 + 1;
    ULINT_LOCAL_AUTO_1 := ULINT_LOCAL_AUTO_1 + 1;
    USINT_LOCAL_AUTO_1 := USINT_LOCAL_AUTO_1 + 1;
    WORD_LOCAL_AUTO_1 := WORD_LOCAL_AUTO_1 + 1;

    BOOL_LOCAL_AUTO_2 := BOOL_LOCAL_AUTO_1;
    BYTE_LOCAL_AUTO_2 := BYTE_LOCAL_AUTO_1;
    DATE_LOCAL_AUTO_2 := DATE_LOCAL_AUTO_1;
    DINT_LOCAL_AUTO_2 := DINT_LOCAL_AUTO_1;
    DWORD_LOCAL_AUTO_2 := DWORD_LOCAL_AUTO_1;
    INT_LOCAL_AUTO_2 := INT_LOCAL_AUTO_1;
    LINT_LOCAL_AUTO_2 := LINT_LOCAL_AUTO_1;
    LREAL_LOCAL_AUTO_2 := LREAL_LOCAL_AUTO_1;
    LWORD_LOCAL_AUTO_2 := LWORD_LOCAL_AUTO_1;
    REAL_LOCAL_AUTO_2 := REAL_LOCAL_AUTO_1;
    SINT_LOCAL_AUTO_2 := SINT_LOCAL_AUTO_1;
    STRING_LOCAL_AUTO_2 := STRING_LOCAL_AUTO_1;
    TIME_LOCAL_AUTO_2 := TIME_LOCAL_AUTO_1;
    UDINT_LOCAL_AUTO_2 := UDINT_LOCAL_AUTO_1;
    UINT_LOCAL_AUTO_2 := UINT_LOCAL_AUTO_1;
    ULINT_LOCAL_AUTO_2 := ULINT_LOCAL_AUTO_1;
    USINT_LOCAL_AUTO_2 := USINT_LOCAL_AUTO_1;
    WORD_LOCAL_AUTO_2 := WORD_LOCAL_AUTO_1;

    // ВЫХОДНЫЕ ПЕРЕМЕННЫЕ
    BOOL_OUT_RETAIN := NOT BOOL_OUT_RETAIN;
    BYTE_OUT_RETAIN := BYTE_OUT_RETAIN + 1;
    DATE_OUT_RETAIN := ANY_TO_DATE(1445385600 + DINT_OUT_RETAIN * 86400);
    DINT_OUT_RETAIN := DINT_OUT_RETAIN + 1;
    DWORD_OUT_RETAIN := DWORD_OUT_RETAIN + 1;
    INT_OUT_RETAIN := INT_OUT_RETAIN + 1;
    LINT_OUT_RETAIN := LINT_OUT_RETAIN + 1;
    LREAL_OUT_RETAIN := LREAL_OUT_RETAIN + 1.1;
    LWORD_OUT_RETAIN := LWORD_OUT_RETAIN + 1;
    REAL_OUT_RETAIN := REAL_OUT_RETAIN + 1.1;
    SINT_OUT_RETAIN := SINT_OUT_RETAIN + 1;
    STRING_OUT_RETAIN := ANY_TO_STRING(DINT_OUT_RETAIN) + ' ' + ANY_TO_STRING(TIME_OUT_RETAIN);
    TIME_OUT_RETAIN := TIME_OUT_RETAIN + T#10s;
    UDINT_OUT_RETAIN := UDINT_OUT_RETAIN + 1;
    UINT_OUT_RETAIN := UINT_OUT_RETAIN + 1;
    ULINT_OUT_RETAIN := ULINT_OUT_RETAIN + 1;
    USINT_OUT_RETAIN := USINT_OUT_RETAIN + 1;
    WORD_OUT_RETAIN := WORD_OUT_RETAIN + 1;

    BOOL_OUT_NON_RETAIN := NOT BOOL_OUT_NON_RETAIN;
    BYTE_OUT_NON_RETAIN := BYTE_OUT_NON_RETAIN + 1;
    DATE_OUT_NON_RETAIN := ANY_TO_DATE(1445385600 + DINT_OUT_NON_RETAIN * 86400);
    DINT_OUT_NON_RETAIN := DINT_OUT_NON_RETAIN + 1;
    DWORD_OUT_NON_RETAIN := DWORD_OUT_NON_RETAIN + 1;
    INT_OUT_NON_RETAIN := INT_OUT_NON_RETAIN + 1;
    LINT_OUT_NON_RETAIN := LINT_OUT_NON_RETAIN + 1;
    LREAL_OUT_NON_RETAIN := LREAL_OUT_NON_RETAIN + 1.1;
    LWORD_OUT_NON_RETAIN := LWORD_OUT_NON_RETAIN + 1;
    REAL_OUT_NON_RETAIN := REAL_OUT_NON_RETAIN + 1.1;
    SINT_OUT_NON_RETAIN := SINT_OUT_NON_RETAIN + 1;
    STRING_OUT_NON_RETAIN := ANY_TO_STRING(DINT_OUT_NON_RETAIN) + ' ' + ANY_TO_STRING(TIME_OUT_NON_RETAIN);
    TIME_OUT_NON_RETAIN := TIME_OUT_NON_RETAIN + T#10s;
    UDINT_OUT_NON_RETAIN := UDINT_OUT_NON_RETAIN + 1;
    UINT_OUT_NON_RETAIN := UINT_OUT_NON_RETAIN + 1;
    ULINT_OUT_NON_RETAIN := ULINT_OUT_NON_RETAIN + 1;
    USINT_OUT_NON_RETAIN := USINT_OUT_NON_RETAIN + 1;
    WORD_OUT_NON_RETAIN := WORD_OUT_NON_RETAIN + 1;

    BOOL_OUT_AUTO_1 := NOT BOOL_OUT_AUTO_1;
    BYTE_OUT_AUTO_1 := BYTE_OUT_AUTO_1 + 1;
    DATE_OUT_AUTO_1 := ANY_TO_DATE(1445385600 + DINT_OUT_AUTO_1 * 86400);
    DINT_OUT_AUTO_1 := DINT_OUT_AUTO_1 + 1;
    DWORD_OUT_AUTO_1 := DWORD_OUT_AUTO_1 + 1;
    INT_OUT_AUTO_1 := INT_OUT_AUTO_1 + 1;
    LINT_OUT_AUTO_1 := LINT_OUT_AUTO_1 + 1;
    LREAL_OUT_AUTO_1 := LREAL_OUT_AUTO_1 + 1.1;
    LWORD_OUT_AUTO_1 := LWORD_OUT_AUTO_1 + 1;
    REAL_OUT_AUTO_1 := REAL_OUT_AUTO_1 + 1.1;
    SINT_OUT_AUTO_1 := SINT_OUT_AUTO_1 + 1;
    STRING_OUT_AUTO_1 := ANY_TO_STRING(DINT_OUT_AUTO_1) + ' ' + ANY_TO_STRING(TIME_OUT_AUTO_1);
    TIME_OUT_AUTO_1 := TIME_OUT_AUTO_1 + T#10s;
    UDINT_OUT_AUTO_1 := UDINT_OUT_AUTO_1 + 1;
    UINT_OUT_AUTO_1 := UINT_OUT_AUTO_1 + 1;
    ULINT_OUT_AUTO_1 := ULINT_OUT_AUTO_1 + 1;
    USINT_OUT_AUTO_1 := USINT_OUT_AUTO_1 + 1;
    WORD_OUT_AUTO_1 := WORD_OUT_AUTO_1 + 1;

    BOOL_OUT_AUTO_2 := BOOL_OUT_AUTO_1;
    BYTE_OUT_AUTO_2 := BYTE_OUT_AUTO_1;
    DATE_OUT_AUTO_2 := DATE_OUT_AUTO_1;
    DINT_OUT_AUTO_2 := DINT_OUT_AUTO_1;
    DWORD_OUT_AUTO_2 := DWORD_OUT_AUTO_1;
    INT_OUT_AUTO_2 := INT_OUT_AUTO_1;
    LINT_OUT_AUTO_2 := LINT_OUT_AUTO_1;
    LREAL_OUT_AUTO_2 := LREAL_OUT_AUTO_1;
    LWORD_OUT_AUTO_2 := LWORD_OUT_AUTO_1;
    REAL_OUT_AUTO_2 := REAL_OUT_AUTO_1;
    SINT_OUT_AUTO_2 := SINT_OUT_AUTO_1;
    STRING_OUT_AUTO_2 := STRING_OUT_AUTO_1;
    TIME_OUT_AUTO_2 := TIME_OUT_AUTO_1;
    UDINT_OUT_AUTO_2 := UDINT_OUT_AUTO_1;
    UINT_OUT_AUTO_2 := UINT_OUT_AUTO_1;
    ULINT_OUT_AUTO_2 := ULINT_OUT_AUTO_1;
    USINT_OUT_AUTO_2 := USINT_OUT_AUTO_1;
    WORD_OUT_AUTO_2 := WORD_OUT_AUTO_1;

END_IF;

END_FUNCTION_BLOCK

(* ---- FB_SIMPLE_TYPE_AUTO.st ---- *)
FUNCTION_BLOCK FB_SIMPLE_TYPE_AUTO_copy

IF TRIGGER_IMP THEN

    BOOL_LOCAL_1 := NOT BOOL_LOCAL_1;
    BYTE_LOCAL_1 := BYTE_LOCAL_1 + 1;
    DATE_LOCAL_1 := ANY_TO_DATE(1445385600 + DINT_LOCAL_1 * 86400);
    DINT_LOCAL_1 := DINT_LOCAL_1 + 1;
    DWORD_LOCAL_1 := DWORD_LOCAL_1 + 1;
    INT_LOCAL_1 := INT_LOCAL_1 + 1;
    LINT_LOCAL_1 := LINT_LOCAL_1 + 1;
    LREAL_LOCAL_1 := LREAL_LOCAL_1 + 1.1;
    LWORD_LOCAL_1 := LWORD_LOCAL_1 + 1;
    REAL_LOCAL_1 := REAL_LOCAL_1 + 1.1;
    SINT_LOCAL_1 := SINT_LOCAL_1 + 1;
    STRING_LOCAL_1 := ANY_TO_STRING(DINT_LOCAL_1) + ' ' + ANY_TO_STRING(TIME_LOCAL_1);
    TIME_LOCAL_1 := TIME_LOCAL_1 + T#10s;
    UDINT_LOCAL_1 := UDINT_LOCAL_1 + 1;
    UINT_LOCAL_1 := UINT_LOCAL_1 + 1;
    ULINT_LOCAL_1 := ULINT_LOCAL_1 + 1;
    USINT_LOCAL_1 := USINT_LOCAL_1 + 1;
    WORD_LOCAL_1 := WORD_LOCAL_1 + 1;

    BOOL_LOCAL_2 := BOOL_LOCAL_1;
    BYTE_LOCAL_2 := BYTE_LOCAL_1;
    DATE_LOCAL_2 := DATE_LOCAL_1;
    DINT_LOCAL_2 := DINT_LOCAL_1;
    DWORD_LOCAL_2 := DWORD_LOCAL_1;
    INT_LOCAL_2 := INT_LOCAL_1;
    LINT_LOCAL_2 := LINT_LOCAL_1;
    LREAL_LOCAL_2 := LREAL_LOCAL_1;
    LWORD_LOCAL_2 := LWORD_LOCAL_1;
    REAL_LOCAL_2 := REAL_LOCAL_1;
    SINT_LOCAL_2 := SINT_LOCAL_1;
    STRING_LOCAL_2 := STRING_LOCAL_1;
    TIME_LOCAL_2 := TIME_LOCAL_1;
    UDINT_LOCAL_2 := UDINT_LOCAL_1;
    UINT_LOCAL_2 := UINT_LOCAL_1;
    ULINT_LOCAL_2 := ULINT_LOCAL_1;
    USINT_LOCAL_2 := USINT_LOCAL_1;
    WORD_LOCAL_2 := WORD_LOCAL_1;

    BOOL_OUT_1 := NOT BOOL_OUT_1;
    BYTE_OUT_1 := BYTE_OUT_1 + 1;
    DATE_OUT_1 := ANY_TO_DATE(1445385600 + DINT_OUT_1 * 86400);
    DINT_OUT_1 := DINT_OUT_1 + 1;
    DWORD_OUT_1 := DWORD_OUT_1 + 1;
    INT_OUT_1 := INT_OUT_1 + 1;
    LINT_OUT_1 := LINT_OUT_1 + 1;
    LREAL_OUT_1 := LREAL_OUT_1 + 1.1;
    LWORD_OUT_1 := LWORD_OUT_1 + 1;
    REAL_OUT_1 := REAL_OUT_1 + 1.1;
    SINT_OUT_1 := SINT_OUT_1 + 1;
    STRING_OUT_1 := ANY_TO_STRING(DINT_OUT_1) + ' ' + ANY_TO_STRING(TIME_OUT_1);
    TIME_OUT_1 := TIME_OUT_1 + T#10s;
    UDINT_OUT_1 := UDINT_OUT_1 + 1;
    UINT_OUT_1 := UINT_OUT_1 + 1;
    ULINT_OUT_1 := ULINT_OUT_1 + 1;
    USINT_OUT_1 := USINT_OUT_1 + 1;
    WORD_OUT_1 := WORD_OUT_1 + 1;

    BOOL_OUT_2 := BOOL_OUT_1;
    BYTE_OUT_2 := BYTE_OUT_1;
    DATE_OUT_2 := DATE_OUT_1;
    DINT_OUT_2 := DINT_OUT_1;
    DWORD_OUT_2 := DWORD_OUT_1;
    INT_OUT_2 := INT_OUT_1;
    LINT_OUT_2 := LINT_OUT_1;
    LREAL_OUT_2 := LREAL_OUT_1;
    LWORD_OUT_2 := LWORD_OUT_1;
    REAL_OUT_2 := REAL_OUT_1;
    SINT_OUT_2 := SINT_OUT_1;
    STRING_OUT_2 := STRING_OUT_1;
    TIME_OUT_2 := TIME_OUT_1;
    UDINT_OUT_2 := UDINT_OUT_1;
    UINT_OUT_2 := UINT_OUT_1;
    ULINT_OUT_2 := ULINT_OUT_1;
    USINT_OUT_2 := USINT_OUT_1;
    WORD_OUT_2 := WORD_OUT_1;

END_IF;

END_FUNCTION_BLOCK

(* ---- FB_SIMPLE_TYPE_NON_RETAIN.st ---- *)
FUNCTION_BLOCK FB_SIMPLE_TYPE_NON_RETAIN

IF TRIGGER_IMP THEN

    BOOL_LOCAL := NOT BOOL_LOCAL;
    BYTE_LOCAL := BYTE_LOCAL + 1;
    DATE_LOCAL := ANY_TO_DATE(1445385600 + DINT_LOCAL * 86400);
    DINT_LOCAL := DINT_LOCAL + 1;
    DWORD_LOCAL := DWORD_LOCAL + 1;
    INT_LOCAL := INT_LOCAL + 1;
    LINT_LOCAL := LINT_LOCAL + 1;
    LREAL_LOCAL := LREAL_LOCAL + 1.1;
    LWORD_LOCAL := LWORD_LOCAL + 1;
    REAL_LOCAL := REAL_LOCAL + 1.1;
    SINT_LOCAL := SINT_LOCAL + 1;
    STRING_LOCAL := ANY_TO_STRING(DINT_LOCAL) + ' ' + ANY_TO_STRING(TIME_LOCAL);
    TIME_LOCAL := TIME_LOCAL + T#10s;
    UDINT_LOCAL := UDINT_LOCAL + 1;
    UINT_LOCAL := UINT_LOCAL + 1;
    ULINT_LOCAL := ULINT_LOCAL + 1;
    USINT_LOCAL := USINT_LOCAL + 1;
    WORD_LOCAL := WORD_LOCAL + 1;

    BOOL_OUT := NOT BOOL_OUT;
    BYTE_OUT := BYTE_OUT + 1;
    DATE_OUT := ANY_TO_DATE(1445385600 + DINT_OUT * 86400);
    DINT_OUT := DINT_OUT + 1;
    DWORD_OUT := DWORD_OUT + 1;
    INT_OUT := INT_OUT + 1;
    LINT_OUT := LINT_OUT + 1;
    LREAL_OUT := LREAL_OUT + 1.1;
    LWORD_OUT := LWORD_OUT + 1;
    REAL_OUT := REAL_OUT + 1.1;
    SINT_OUT := SINT_OUT + 1;
    STRING_OUT := ANY_TO_STRING(DINT_OUT) + ' ' + ANY_TO_STRING(TIME_OUT);
    TIME_OUT := TIME_OUT + T#10s;
    UDINT_OUT := UDINT_OUT + 1;
    UINT_OUT := UINT_OUT + 1;
    ULINT_OUT := ULINT_OUT + 1;
    USINT_OUT := USINT_OUT + 1;
    WORD_OUT := WORD_OUT + 1;

END_IF;

END_FUNCTION_BLOCK

(* ---- FB_SIMPLE_TYPE_RETAIN.st ---- *)
FUNCTION_BLOCK FB_SIMPLE_TYPE_RETAIN

IF TRIGGER_IMP THEN

    BOOL_LOCAL := NOT BOOL_LOCAL;
    BYTE_LOCAL := BYTE_LOCAL + 1;
    DATE_LOCAL := ANY_TO_DATE(1445385600 + DINT_LOCAL * 86400);
    DINT_LOCAL := DINT_LOCAL + 1;
    DWORD_LOCAL := DWORD_LOCAL + 1;
    INT_LOCAL := INT_LOCAL + 1;
    LINT_LOCAL := LINT_LOCAL + 1;
    LREAL_LOCAL := LREAL_LOCAL + 1.1;
    LWORD_LOCAL := LWORD_LOCAL + 1;
    REAL_LOCAL := REAL_LOCAL + 1.1;
    SINT_LOCAL := SINT_LOCAL + 1;
    STRING_LOCAL := ANY_TO_STRING(DINT_LOCAL) + ' ' + ANY_TO_STRING(TIME_LOCAL);
    TIME_LOCAL := TIME_LOCAL + T#10s;
    UDINT_LOCAL := UDINT_LOCAL + 1;
    UINT_LOCAL := UINT_LOCAL + 1;
    ULINT_LOCAL := ULINT_LOCAL + 1;
    USINT_LOCAL := USINT_LOCAL + 1;
    WORD_LOCAL := WORD_LOCAL + 1;

    BOOL_OUT := NOT BOOL_OUT;
    BYTE_OUT := BYTE_OUT + 1;
    DATE_OUT := ANY_TO_DATE(1445385600 + DINT_OUT * 86400);
    DINT_OUT := DINT_OUT + 1;
    DWORD_OUT := DWORD_OUT + 1;
    INT_OUT := INT_OUT + 1;
    LINT_OUT := LINT_OUT + 1;
    LREAL_OUT := LREAL_OUT + 1.1;
    LWORD_OUT := LWORD_OUT + 1;
    REAL_OUT := REAL_OUT + 1.1;
    SINT_OUT := SINT_OUT + 1;
    STRING_OUT := ANY_TO_STRING(DINT_OUT) + ' ' + ANY_TO_STRING(TIME_OUT);
    TIME_OUT := TIME_OUT + T#10s;
    UDINT_OUT := UDINT_OUT + 1;
    UINT_OUT := UINT_OUT + 1;
    ULINT_OUT := ULINT_OUT + 1;
    USINT_OUT := USINT_OUT + 1;
    WORD_OUT := WORD_OUT + 1;

END_IF;

END_FUNCTION_BLOCK

(* ---- FB_STRUCTURE_SIMPLE_TYPE.st ---- *)
FUNCTION_BLOCK FB_STRUCTURE_SIMPLE_TYPE

IF TRIGGER_IMP THEN

    // ЛОКАЛЬНЫЕ ПЕРЕМЕННЫЕ
    STRUCTURE_LOCAL_RETAIN.BOOL_TYPE := NOT STRUCTURE_LOCAL_RETAIN.BOOL_TYPE;
    STRUCTURE_LOCAL_RETAIN.BYTE_TYPE := STRUCTURE_LOCAL_RETAIN.BYTE_TYPE + 1;
    STRUCTURE_LOCAL_RETAIN.DATE_TYPE := ANY_TO_DATE(1445385600 + STRUCTURE_LOCAL_RETAIN.DINT_TYPE * 86400);
    STRUCTURE_LOCAL_RETAIN.DINT_TYPE := STRUCTURE_LOCAL_RETAIN.DINT_TYPE + 1;
    STRUCTURE_LOCAL_RETAIN.DWORD_TYPE := STRUCTURE_LOCAL_RETAIN.DWORD_TYPE + 1;
    STRUCTURE_LOCAL_RETAIN.INT_TYPE := STRUCTURE_LOCAL_RETAIN.INT_TYPE + 1;
    STRUCTURE_LOCAL_RETAIN.LINT_TYPE := STRUCTURE_LOCAL_RETAIN.LINT_TYPE + 1;
    STRUCTURE_LOCAL_RETAIN.LREAL_TYPE := STRUCTURE_LOCAL_RETAIN.LREAL_TYPE + 1;
    STRUCTURE_LOCAL_RETAIN.LWORD_TYPE := STRUCTURE_LOCAL_RETAIN.LWORD_TYPE + 1;
    STRUCTURE_LOCAL_RETAIN.REAL_TYPE := STRUCTURE_LOCAL_RETAIN.REAL_TYPE + 1;
    STRUCTURE_LOCAL_RETAIN.SINT_TYPE := STRUCTURE_LOCAL_RETAIN.SINT_TYPE + 1;
    STRUCTURE_LOCAL_RETAIN.STRING_TYPE := ANY_TO_STRING(STRUCTURE_LOCAL_RETAIN.DINT_TYPE) + ' ' + ANY_TO_STRING(STRUCTURE_LOCAL_RETAIN.TIME_TYPE);
    STRUCTURE_LOCAL_RETAIN.TIME_TYPE := STRUCTURE_LOCAL_RETAIN.TIME_TYPE + PULSE_TIME;
    STRUCTURE_LOCAL_RETAIN.UDINT_TYPE := STRUCTURE_LOCAL_RETAIN.UDINT_TYPE + 1;
    STRUCTURE_LOCAL_RETAIN.UINT_TYPE := STRUCTURE_LOCAL_RETAIN.UINT_TYPE + 1;
    STRUCTURE_LOCAL_RETAIN.ULINT_TYPE := STRUCTURE_LOCAL_RETAIN.ULINT_TYPE + 1;
    STRUCTURE_LOCAL_RETAIN.USINT_TYPE := STRUCTURE_LOCAL_RETAIN.USINT_TYPE + 1;
    STRUCTURE_LOCAL_RETAIN.WORD_TYPE := STRUCTURE_LOCAL_RETAIN.WORD_TYPE + 1;

    STRUCTURE_LOCAL_NON_RETAIN.BOOL_TYPE := NOT STRUCTURE_LOCAL_NON_RETAIN.BOOL_TYPE;
    STRUCTURE_LOCAL_NON_RETAIN.BYTE_TYPE := STRUCTURE_LOCAL_NON_RETAIN.BYTE_TYPE + 1;
    STRUCTURE_LOCAL_NON_RETAIN.DATE_TYPE := ANY_TO_DATE(1445385600 + STRUCTURE_LOCAL_NON_RETAIN.DINT_TYPE * 86400);
    STRUCTURE_LOCAL_NON_RETAIN.DINT_TYPE := STRUCTURE_LOCAL_NON_RETAIN.DINT_TYPE + 1;
    STRUCTURE_LOCAL_NON_RETAIN.DWORD_TYPE := STRUCTURE_LOCAL_NON_RETAIN.DWORD_TYPE + 1;
    STRUCTURE_LOCAL_NON_RETAIN.INT_TYPE := STRUCTURE_LOCAL_NON_RETAIN.INT_TYPE + 1;
    STRUCTURE_LOCAL_NON_RETAIN.LINT_TYPE := STRUCTURE_LOCAL_NON_RETAIN.LINT_TYPE + 1;
    STRUCTURE_LOCAL_NON_RETAIN.LREAL_TYPE := STRUCTURE_LOCAL_NON_RETAIN.LREAL_TYPE + 1;
    STRUCTURE_LOCAL_NON_RETAIN.LWORD_TYPE := STRUCTURE_LOCAL_NON_RETAIN.LWORD_TYPE + 1;
    STRUCTURE_LOCAL_NON_RETAIN.REAL_TYPE := STRUCTURE_LOCAL_NON_RETAIN.REAL_TYPE + 1;
    STRUCTURE_LOCAL_NON_RETAIN.SINT_TYPE := STRUCTURE_LOCAL_NON_RETAIN.SINT_TYPE + 1;
    STRUCTURE_LOCAL_NON_RETAIN.STRING_TYPE := ANY_TO_STRING(STRUCTURE_LOCAL_NON_RETAIN.DINT_TYPE) + ' ' + ANY_TO_STRING(STRUCTURE_LOCAL_NON_RETAIN.TIME_TYPE);
    STRUCTURE_LOCAL_NON_RETAIN.TIME_TYPE := STRUCTURE_LOCAL_NON_RETAIN.TIME_TYPE + PULSE_TIME;
    STRUCTURE_LOCAL_NON_RETAIN.UDINT_TYPE := STRUCTURE_LOCAL_NON_RETAIN.UDINT_TYPE + 1;
    STRUCTURE_LOCAL_NON_RETAIN.UINT_TYPE := STRUCTURE_LOCAL_NON_RETAIN.UINT_TYPE + 1;
    STRUCTURE_LOCAL_NON_RETAIN.ULINT_TYPE := STRUCTURE_LOCAL_NON_RETAIN.ULINT_TYPE + 1;
    STRUCTURE_LOCAL_NON_RETAIN.USINT_TYPE := STRUCTURE_LOCAL_NON_RETAIN.USINT_TYPE + 1;
    STRUCTURE_LOCAL_NON_RETAIN.WORD_TYPE := STRUCTURE_LOCAL_NON_RETAIN.WORD_TYPE + 1;

    STRUCTURE_LOCAL_AUTO_1.BOOL_TYPE := NOT STRUCTURE_LOCAL_AUTO_1.BOOL_TYPE;
    STRUCTURE_LOCAL_AUTO_1.BYTE_TYPE := STRUCTURE_LOCAL_AUTO_1.BYTE_TYPE + 1;
    STRUCTURE_LOCAL_AUTO_1.DATE_TYPE := ANY_TO_DATE(1445385600 + STRUCTURE_LOCAL_AUTO_1.DINT_TYPE * 86400);
    STRUCTURE_LOCAL_AUTO_1.DINT_TYPE := STRUCTURE_LOCAL_AUTO_1.DINT_TYPE + 1;
    STRUCTURE_LOCAL_AUTO_1.DWORD_TYPE := STRUCTURE_LOCAL_AUTO_1.DWORD_TYPE + 1;
    STRUCTURE_LOCAL_AUTO_1.INT_TYPE := STRUCTURE_LOCAL_AUTO_1.INT_TYPE + 1;
    STRUCTURE_LOCAL_AUTO_1.LINT_TYPE := STRUCTURE_LOCAL_AUTO_1.LINT_TYPE + 1;
    STRUCTURE_LOCAL_AUTO_1.LREAL_TYPE := STRUCTURE_LOCAL_AUTO_1.LREAL_TYPE + 1;
    STRUCTURE_LOCAL_AUTO_1.LWORD_TYPE := STRUCTURE_LOCAL_AUTO_1.LWORD_TYPE + 1;
    STRUCTURE_LOCAL_AUTO_1.REAL_TYPE := STRUCTURE_LOCAL_AUTO_1.REAL_TYPE + 1;
    STRUCTURE_LOCAL_AUTO_1.SINT_TYPE := STRUCTURE_LOCAL_AUTO_1.SINT_TYPE + 1;
    STRUCTURE_LOCAL_AUTO_1.STRING_TYPE := ANY_TO_STRING(STRUCTURE_LOCAL_AUTO_1.DINT_TYPE) + ' ' + ANY_TO_STRING(STRUCTURE_LOCAL_AUTO_1.TIME_TYPE);
    STRUCTURE_LOCAL_AUTO_1.TIME_TYPE := STRUCTURE_LOCAL_AUTO_1.TIME_TYPE + PULSE_TIME;
    STRUCTURE_LOCAL_AUTO_1.UDINT_TYPE := STRUCTURE_LOCAL_AUTO_1.UDINT_TYPE + 1;
    STRUCTURE_LOCAL_AUTO_1.UINT_TYPE := STRUCTURE_LOCAL_AUTO_1.UINT_TYPE + 1;
    STRUCTURE_LOCAL_AUTO_1.ULINT_TYPE := STRUCTURE_LOCAL_AUTO_1.ULINT_TYPE + 1;
    STRUCTURE_LOCAL_AUTO_1.USINT_TYPE := STRUCTURE_LOCAL_AUTO_1.USINT_TYPE + 1;
    STRUCTURE_LOCAL_AUTO_1.WORD_TYPE := STRUCTURE_LOCAL_AUTO_1.WORD_TYPE + 1;

    STRUCTURE_LOCAL_AUTO_2.BOOL_TYPE := STRUCTURE_LOCAL_AUTO_1.BOOL_TYPE;
    STRUCTURE_LOCAL_AUTO_2.BYTE_TYPE := STRUCTURE_LOCAL_AUTO_1.BYTE_TYPE;
    STRUCTURE_LOCAL_AUTO_2.DATE_TYPE := STRUCTURE_LOCAL_AUTO_1.DATE_TYPE;
    STRUCTURE_LOCAL_AUTO_2.DINT_TYPE := STRUCTURE_LOCAL_AUTO_1.DINT_TYPE;
    STRUCTURE_LOCAL_AUTO_2.DWORD_TYPE := STRUCTURE_LOCAL_AUTO_1.DWORD_TYPE;
    STRUCTURE_LOCAL_AUTO_2.INT_TYPE := STRUCTURE_LOCAL_AUTO_1.INT_TYPE;
    STRUCTURE_LOCAL_AUTO_2.LINT_TYPE := STRUCTURE_LOCAL_AUTO_1.LINT_TYPE;
    STRUCTURE_LOCAL_AUTO_2.LREAL_TYPE := STRUCTURE_LOCAL_AUTO_1.LREAL_TYPE;
    STRUCTURE_LOCAL_AUTO_2.LWORD_TYPE := STRUCTURE_LOCAL_AUTO_1.LWORD_TYPE;
    STRUCTURE_LOCAL_AUTO_2.REAL_TYPE := STRUCTURE_LOCAL_AUTO_1.REAL_TYPE;
    STRUCTURE_LOCAL_AUTO_2.SINT_TYPE := STRUCTURE_LOCAL_AUTO_1.SINT_TYPE;
    STRUCTURE_LOCAL_AUTO_2.STRING_TYPE := STRUCTURE_LOCAL_AUTO_1.STRING_TYPE;
    STRUCTURE_LOCAL_AUTO_2.TIME_TYPE := STRUCTURE_LOCAL_AUTO_1.TIME_TYPE;
    STRUCTURE_LOCAL_AUTO_2.UDINT_TYPE := STRUCTURE_LOCAL_AUTO_1.UDINT_TYPE;
    STRUCTURE_LOCAL_AUTO_2.UINT_TYPE := STRUCTURE_LOCAL_AUTO_1.UINT_TYPE;
    STRUCTURE_LOCAL_AUTO_2.ULINT_TYPE := STRUCTURE_LOCAL_AUTO_1.ULINT_TYPE;
    STRUCTURE_LOCAL_AUTO_2.USINT_TYPE := STRUCTURE_LOCAL_AUTO_1.USINT_TYPE;
    STRUCTURE_LOCAL_AUTO_2.WORD_TYPE := STRUCTURE_LOCAL_AUTO_1.WORD_TYPE;

    // ВЫХОДНЫЕ ПЕРЕМЕННЫЕ
    STRUCTURE_OUT_RETAIN.BOOL_TYPE := NOT STRUCTURE_OUT_RETAIN.BOOL_TYPE;
    STRUCTURE_OUT_RETAIN.BYTE_TYPE := STRUCTURE_OUT_RETAIN.BYTE_TYPE + 1;
    STRUCTURE_OUT_RETAIN.DATE_TYPE := ANY_TO_DATE(1445385600 + STRUCTURE_OUT_RETAIN.DINT_TYPE * 86400);
    STRUCTURE_OUT_RETAIN.DINT_TYPE := STRUCTURE_OUT_RETAIN.DINT_TYPE + 1;
    STRUCTURE_OUT_RETAIN.DWORD_TYPE := STRUCTURE_OUT_RETAIN.DWORD_TYPE + 1;
    STRUCTURE_OUT_RETAIN.INT_TYPE := STRUCTURE_OUT_RETAIN.INT_TYPE + 1;
    STRUCTURE_OUT_RETAIN.LINT_TYPE := STRUCTURE_OUT_RETAIN.LINT_TYPE + 1;
    STRUCTURE_OUT_RETAIN.LREAL_TYPE := STRUCTURE_OUT_RETAIN.LREAL_TYPE + 1;
    STRUCTURE_OUT_RETAIN.LWORD_TYPE := STRUCTURE_OUT_RETAIN.LWORD_TYPE + 1;
    STRUCTURE_OUT_RETAIN.REAL_TYPE := STRUCTURE_OUT_RETAIN.REAL_TYPE + 1;
    STRUCTURE_OUT_RETAIN.SINT_TYPE := STRUCTURE_OUT_RETAIN.SINT_TYPE + 1;
    STRUCTURE_OUT_RETAIN.STRING_TYPE := ANY_TO_STRING(STRUCTURE_OUT_RETAIN.DINT_TYPE) + ' ' + ANY_TO_STRING(STRUCTURE_OUT_RETAIN.TIME_TYPE);
    STRUCTURE_OUT_RETAIN.TIME_TYPE := STRUCTURE_OUT_RETAIN.TIME_TYPE + PULSE_TIME;
    STRUCTURE_OUT_RETAIN.UDINT_TYPE := STRUCTURE_OUT_RETAIN.UDINT_TYPE + 1;
    STRUCTURE_OUT_RETAIN.UINT_TYPE := STRUCTURE_OUT_RETAIN.UINT_TYPE + 1;
    STRUCTURE_OUT_RETAIN.ULINT_TYPE := STRUCTURE_OUT_RETAIN.ULINT_TYPE + 1;
    STRUCTURE_OUT_RETAIN.USINT_TYPE := STRUCTURE_OUT_RETAIN.USINT_TYPE + 1;
    STRUCTURE_OUT_RETAIN.WORD_TYPE := STRUCTURE_OUT_RETAIN.WORD_TYPE + 1;

    STRUCTURE_OUT_NON_RETAIN.BOOL_TYPE := NOT STRUCTURE_OUT_NON_RETAIN.BOOL_TYPE;
    STRUCTURE_OUT_NON_RETAIN.BYTE_TYPE := STRUCTURE_OUT_NON_RETAIN.BYTE_TYPE + 1;
    STRUCTURE_OUT_NON_RETAIN.DATE_TYPE := ANY_TO_DATE(1445385600 + STRUCTURE_OUT_NON_RETAIN.DINT_TYPE * 86400);
    STRUCTURE_OUT_NON_RETAIN.DINT_TYPE := STRUCTURE_OUT_NON_RETAIN.DINT_TYPE + 1;
    STRUCTURE_OUT_NON_RETAIN.DWORD_TYPE := STRUCTURE_OUT_NON_RETAIN.DWORD_TYPE + 1;
    STRUCTURE_OUT_NON_RETAIN.INT_TYPE := STRUCTURE_OUT_NON_RETAIN.INT_TYPE + 1;
    STRUCTURE_OUT_NON_RETAIN.LINT_TYPE := STRUCTURE_OUT_NON_RETAIN.LINT_TYPE + 1;
    STRUCTURE_OUT_NON_RETAIN.LREAL_TYPE := STRUCTURE_OUT_NON_RETAIN.LREAL_TYPE + 1;
    STRUCTURE_OUT_NON_RETAIN.LWORD_TYPE := STRUCTURE_OUT_NON_RETAIN.LWORD_TYPE + 1;
    STRUCTURE_OUT_NON_RETAIN.REAL_TYPE := STRUCTURE_OUT_NON_RETAIN.REAL_TYPE + 1;
    STRUCTURE_OUT_NON_RETAIN.SINT_TYPE := STRUCTURE_OUT_NON_RETAIN.SINT_TYPE + 1;
    STRUCTURE_OUT_NON_RETAIN.STRING_TYPE := ANY_TO_STRING(STRUCTURE_OUT_NON_RETAIN.DINT_TYPE) + ' ' + ANY_TO_STRING(STRUCTURE_OUT_NON_RETAIN.TIME_TYPE);
    STRUCTURE_OUT_NON_RETAIN.TIME_TYPE := STRUCTURE_OUT_NON_RETAIN.TIME_TYPE + PULSE_TIME;
    STRUCTURE_OUT_NON_RETAIN.UDINT_TYPE := STRUCTURE_OUT_NON_RETAIN.UDINT_TYPE + 1;
    STRUCTURE_OUT_NON_RETAIN.UINT_TYPE := STRUCTURE_OUT_NON_RETAIN.UINT_TYPE + 1;
    STRUCTURE_OUT_NON_RETAIN.ULINT_TYPE := STRUCTURE_OUT_NON_RETAIN.ULINT_TYPE + 1;
    STRUCTURE_OUT_NON_RETAIN.USINT_TYPE := STRUCTURE_OUT_NON_RETAIN.USINT_TYPE + 1;
    STRUCTURE_OUT_NON_RETAIN.WORD_TYPE := STRUCTURE_OUT_NON_RETAIN.WORD_TYPE + 1;

    STRUCTURE_OUT_AUTO_1.BOOL_TYPE := NOT STRUCTURE_OUT_AUTO_1.BOOL_TYPE;
    STRUCTURE_OUT_AUTO_1.BYTE_TYPE := STRUCTURE_OUT_AUTO_1.BYTE_TYPE + 1;
    STRUCTURE_OUT_AUTO_1.DATE_TYPE := ANY_TO_DATE(1445385600 + STRUCTURE_OUT_AUTO_1.DINT_TYPE * 86400);
    STRUCTURE_OUT_AUTO_1.DINT_TYPE := STRUCTURE_OUT_AUTO_1.DINT_TYPE + 1;
    STRUCTURE_OUT_AUTO_1.DWORD_TYPE := STRUCTURE_OUT_AUTO_1.DWORD_TYPE + 1;
    STRUCTURE_OUT_AUTO_1.INT_TYPE := STRUCTURE_OUT_AUTO_1.INT_TYPE + 1;
    STRUCTURE_OUT_AUTO_1.LINT_TYPE := STRUCTURE_OUT_AUTO_1.LINT_TYPE + 1;
    STRUCTURE_OUT_AUTO_1.LREAL_TYPE := STRUCTURE_OUT_AUTO_1.LREAL_TYPE + 1;
    STRUCTURE_OUT_AUTO_1.LWORD_TYPE := STRUCTURE_OUT_AUTO_1.LWORD_TYPE + 1;
    STRUCTURE_OUT_AUTO_1.REAL_TYPE := STRUCTURE_OUT_AUTO_1.REAL_TYPE + 1;
    STRUCTURE_OUT_AUTO_1.SINT_TYPE := STRUCTURE_OUT_AUTO_1.SINT_TYPE + 1;
    STRUCTURE_OUT_AUTO_1.STRING_TYPE := ANY_TO_STRING(STRUCTURE_OUT_AUTO_1.DINT_TYPE) + ' ' + ANY_TO_STRING(STRUCTURE_OUT_AUTO_1.TIME_TYPE);
    STRUCTURE_OUT_AUTO_1.TIME_TYPE := STRUCTURE_OUT_AUTO_1.TIME_TYPE + PULSE_TIME;
    STRUCTURE_OUT_AUTO_1.UDINT_TYPE := STRUCTURE_OUT_AUTO_1.UDINT_TYPE + 1;
    STRUCTURE_OUT_AUTO_1.UINT_TYPE := STRUCTURE_OUT_AUTO_1.UINT_TYPE + 1;
    STRUCTURE_OUT_AUTO_1.ULINT_TYPE := STRUCTURE_OUT_AUTO_1.ULINT_TYPE + 1;
    STRUCTURE_OUT_AUTO_1.USINT_TYPE := STRUCTURE_OUT_AUTO_1.USINT_TYPE + 1;
    STRUCTURE_OUT_AUTO_1.WORD_TYPE := STRUCTURE_OUT_AUTO_1.WORD_TYPE + 1;

    STRUCTURE_OUT_AUTO_2.BOOL_TYPE := STRUCTURE_OUT_AUTO_1.BOOL_TYPE;
    STRUCTURE_OUT_AUTO_2.BYTE_TYPE := STRUCTURE_OUT_AUTO_1.BYTE_TYPE;
    STRUCTURE_OUT_AUTO_2.DATE_TYPE := STRUCTURE_OUT_AUTO_1.DATE_TYPE;
    STRUCTURE_OUT_AUTO_2.DINT_TYPE := STRUCTURE_OUT_AUTO_1.DINT_TYPE;
    STRUCTURE_OUT_AUTO_2.DWORD_TYPE := STRUCTURE_OUT_AUTO_1.DWORD_TYPE;
    STRUCTURE_OUT_AUTO_2.INT_TYPE := STRUCTURE_OUT_AUTO_1.INT_TYPE;
    STRUCTURE_OUT_AUTO_2.LINT_TYPE := STRUCTURE_OUT_AUTO_1.LINT_TYPE;
    STRUCTURE_OUT_AUTO_2.LREAL_TYPE := STRUCTURE_OUT_AUTO_1.LREAL_TYPE;
    STRUCTURE_OUT_AUTO_2.LWORD_TYPE := STRUCTURE_OUT_AUTO_1.LWORD_TYPE;
    STRUCTURE_OUT_AUTO_2.REAL_TYPE := STRUCTURE_OUT_AUTO_1.REAL_TYPE;
    STRUCTURE_OUT_AUTO_2.SINT_TYPE := STRUCTURE_OUT_AUTO_1.SINT_TYPE;
    STRUCTURE_OUT_AUTO_2.STRING_TYPE := STRUCTURE_OUT_AUTO_1.STRING_TYPE;
    STRUCTURE_OUT_AUTO_2.TIME_TYPE := STRUCTURE_OUT_AUTO_1.TIME_TYPE;
    STRUCTURE_OUT_AUTO_2.UDINT_TYPE := STRUCTURE_OUT_AUTO_1.UDINT_TYPE;
    STRUCTURE_OUT_AUTO_2.UINT_TYPE := STRUCTURE_OUT_AUTO_1.UINT_TYPE;
    STRUCTURE_OUT_AUTO_2.ULINT_TYPE := STRUCTURE_OUT_AUTO_1.ULINT_TYPE;
    STRUCTURE_OUT_AUTO_2.USINT_TYPE := STRUCTURE_OUT_AUTO_1.USINT_TYPE;
    STRUCTURE_OUT_AUTO_2.WORD_TYPE := STRUCTURE_OUT_AUTO_1.WORD_TYPE;

END_IF;

END_FUNCTION_BLOCK
